// TIA Portal V18 export
TYPE "Alarm_ShW"
// stored: IsFailsafeCompliant false
   STRUCT
      Cylinder : Bool;
      Global : Bool;
      Servo : Bool;
      LaserWelding : Bool;
      LaserMarker : Bool;
      Camera : Bool;
      Scanner : Bool;
      RFID : Bool;
      IPC : Bool;
      LeakTester : Bool;
      ScrewDriver : Bool;
      PressingMonitor : Bool;
      Conveyor : Bool;
      Magnetizer : Bool;
      "PLC Connection" : Bool;
   END_STRUCT;
END_TYPE
